(* CODESYS project PLC_CanIftHelper0.0.1.12.library
   Author: Cameron Johnson
   Placeholder: CanItfHelper
   Title: CanItfHelper
   Version: 0.0.1.12
   Description: This library has been supplied by Beckhoff Automation LLC As-Is and is intended only as an example implementation. Functionality is not guaranteed.
   Company: Beckhoff Automation LLC

Project tree, tasks and I/O mapping:
  libraries: Tc2_Standard, * (Beckhoff Automation GmbH); Tc2_System, * (Beckhoff Automation GmbH); Tc2_Utilities, * (Beckhoff Automation GmbH); Tc3_Module, * (Beckhoff Automation GmbH)
  11BitIdentifier/
    DUTs/
      data type ST_CanData_11bit
      data type ST_RxCanQueue_11bit
      data type ST_TxCanQueue_11bit
    POUs/
      function F_HwGetAddrInfo_11bit [ST]
      function F_HwSetAddrInfo_11bit [ST]
  29BitIdentifier/
    DUTs/
      data type ST_CanData_29bit
      data type ST_RxCanQueue_29bit
      data type ST_TxCanQueue_29bit
    POUs/
      function F_HwGetAddrInfo_29bit [ST]
      function F_HwSetAddrInfo_29bit [ST]
  29BitIdentifier_nTranscation/
    DUTs/
      data type ST_CanData_29bit_nTrans
      data type ST_RxCanQueue_29bit_nTrans
      data type ST_TxCanQueue_29bit_nTrans
    POUs/
      function F_HwGetAddrInfo_29bit_nTrans [ST]
      function F_HwSetAddrInfo_29bit_nTrans [ST]
  CanIftHelper/
    DUTs/
      data type E_CanItfHelperHResult
      data type ST_CanHeader
      data type ST_CanMsg
      data type U_RxQueue
      data type U_TxQueue
    POUs/
      function block FB_CanItfHelper [ST]: mCheckSetup, mRxMessageGet, mRxMessagesAck, mTxMessageAdd, mTxMessgesSend, mTxQueueReset
  DUTs/
    data type ST_CanMasterCycleInfo
    data type ST_CanMasterGlobalState
  GVLs/
    global variables GVL_CanItfHelper
    global variables Param_CanItfHelper
  Utilities/
    DUTs/
      data type E_CanRxMapperHResult
      data type ST_RxMapping
    POUs/
      function F_CanMessage_TO_CSV [ST]
      function F_CSV_TO_CanMessage [ST]
      function block FB_RxMapper [ST]: mAddMapping, mCheckSetup, mClearMappings, mCreateMsgMapping, mCreateNewMapping, mSetMappingCnt
  Version/
    global variables Global_Version
*)

// 11BitIdentifier/DUTs/ST_CanData_11bit
{attribute 'pack_mode' := '1'}
TYPE ST_CanData_11bit :
STRUCT
	nCobid: WORD; //bits 0-3 is CAN data length, bit 4 is CAN RTR flag, bit 5-15 is CAN Cobid.
	aData: ARRAY[0..7] OF BYTE;
END_STRUCT
END_TYPE

// 11BitIdentifier/DUTs/ST_RxCanQueue_11bit
{attribute 'pack_mode' := '1'}
TYPE ST_RxCanQueue_11bit :
STRUCT
	nTxCounter: UINT; // Tx handshake
	nRxCounter: UINT; // Rx handshake
	nNoOfmessages: UINT; // Number of messages relevent in Queue, ignore the rest.
	aMessages: ARRAY[0..GVL_CanItfHelper.nRxQueueUpperIndex] OF ST_CanData_11bit;
END_STRUCT
END_TYPE

// 11BitIdentifier/DUTs/ST_TxCanQueue_11bit
{attribute 'pack_mode' := '1'}
TYPE ST_TxCanQueue_11bit :
STRUCT
	nTxCounter: UINT; // Tx handshake
	nRxCounter: UINT; // Rx handshake
	nNoOfmessages: UINT; // Number of messages relevent in Queue, ignore the rest.
	aMessages: ARRAY[0..GVL_CanItfHelper.nTxQueueUpperIndex] OF ST_CanData_11bit;
END_STRUCT
END_TYPE

// 29BitIdentifier/DUTs/ST_CanData_29bit
{attribute 'pack_mode' := '1'}
TYPE ST_CanData_29bit :
STRUCT
	nLength: UINT; //values 0-8
	nCobid: DWORD; // bits0-28 CAN Cobid; bit 30 CAN RTR flag; bit 31 clear -> 11bit CAN Indentifier, set -> 29bit CAN Indentifier.
	aData: ARRAY[0..7] OF BYTE;
END_STRUCT
END_TYPE

// 29BitIdentifier/DUTs/ST_RxCanQueue_29bit
{attribute 'pack_mode' := '1'}
TYPE ST_RxCanQueue_29bit :
STRUCT
	nTxCounter: UINT; // Tx Handshake
	nRxCounter: UINT; // Rx handshake
	nNoOfmessages: UINT; // Number of messages relevent in Queue, ignore the rest.
	aMessages: ARRAY[0..GVL_CanItfHelper.nRxQueueUpperIndex] OF ST_CanData_29bit;
END_STRUCT
END_TYPE

// 29BitIdentifier/DUTs/ST_TxCanQueue_29bit
{attribute 'pack_mode' := '1'}
TYPE ST_TxCanQueue_29bit :
STRUCT
	nTxCounter: UINT; // Tx Handshake
	nRxCounter: UINT; // Rx handshake
	nNoOfmessages: UINT; // Number of messages relevent in Queue, ignore the rest.
	aMessages: ARRAY[0..GVL_CanItfHelper.nTxQueueUpperIndex] OF ST_CanData_29bit;
END_STRUCT
END_TYPE

// 29BitIdentifier_nTranscation/DUTs/ST_CanData_29bit_nTrans
{attribute 'pack_mode' := '1'}
TYPE ST_CanData_29bit_nTrans : //used with CX2500_M510 hardware
STRUCT
	ntransactionNumber : UINT; //unique identifier for message. See TxRxCanQueue.nTranactionNumber to see last TxMsg sent. Not used by FB_CanItfHelper.
	nLength: UINT; //values 0-8
	nCobid: DWORD; // bits0-28 CAN Cobid; bit 30 CAN RTR flag; bit 31 clear -> 11bit CAN Indentifier, set -> 29bit CAN Indentifier.
	aData: ARRAY[0..7] OF BYTE;
END_STRUCT
END_TYPE

// 29BitIdentifier_nTranscation/DUTs/ST_RxCanQueue_29bit_nTrans
{attribute 'pack_mode' := '1'}
TYPE ST_RxCanQueue_29bit_nTrans :
STRUCT
	nTxCounter: UINT; // Tx Handshake
	nRxCounter: UINT; // Rx handshake
	nNoOfmessages: UINT; // Number of messages relevent in Queue, ignore the rest.
	nTranactionNumber : UINT; // nTrans number of last sent TxMsg. Not used by FB_CanItfHelper.
	aMessages: ARRAY[0..GVL_CanItfHelper.nRxQueueUpperIndex] OF ST_CanData_29bit_nTrans;
END_STRUCT
END_TYPE

// 29BitIdentifier_nTranscation/DUTs/ST_TxCanQueue_29bit_nTrans
{attribute 'pack_mode' := '1'}
TYPE ST_TxCanQueue_29bit_nTrans :
STRUCT
	nTxCounter: UINT; 		// Tx Handshake
	nRxCounter: UINT; 		// Rx handshake
	nNoOfmessages: UINT; 	// Number of messages relevent in Queue, ignore the rest.
	nDummy : UINT;			//Reserved
	aMessages: ARRAY[0..GVL_CanItfHelper.nTxQueueUpperIndex] OF ST_CanData_29bit_nTrans;
END_STRUCT
END_TYPE

// CanIftHelper/DUTs/E_CanItfHelperHResult
{attribute 'qualified_only'}
{attribute 'strict'}
TYPE E_CanItfHelperHResult :
(
	NoError 						:= 0,  // values >= 0 implies no error and/or informational. values < 0 implies error. 
	NoError_11Bit					:= 1,
	NoError_29Bit					:= 2,
	NoError_29Bit_nTrans			:= 3,
	
	Error							:= -1, //Error, generic
	InvalidSetup 					:= -2, //pointers to ST_CanQueue are zero or sizeof ST_CanQueue doesn't equal 11bit or 29bit version.
	InvalidPointer					:= -3, //pointer parameter is zero.
	
	RxQueueHasUnreadMessages 		:= -100, // Rx Queue 'NoOfRxMessages' not equal RxMessagesAckedCnt, call either mGetRxMessages or mAckRxMessages.
	RxQueueEmpty 					:= -101, // Rx queue is empty, wait for more data.
	NoNewRxMessages 				:= -102, // Rx queue has not received new data yet.
	RxMessageInvalid				:= -103, // Rx Message returned is invalid, ignore result. Re-read Rx Messages.

	TxQueueFull 					:= -200, //NumOfMessages variable in Tx Queue is at or is greater then the allowed amount. Call aResetTxQueue and refill queue.
	TxQueueEmpty 					:= -201, // Tx queue 'NoOfTxMessages' value is zero, use mAddTxMessage to add messages.
	TxQueueInvalid					:= -202, //Tx Queue
	TxQueueIsBusy					:= -203 // Tx queue 'TxCounter' and Rx queue 'TxCounter' are not equal, waiting for CanInterface to send previous messages.
	
)DINT;
END_TYPE

// CanIftHelper/DUTs/ST_CanHeader
TYPE ST_CanHeader :
STRUCT
	nCobid: DWORD; // User level Cobid, use functions to handle bit mapping to CAN interface process data.
	bExtendedAddress: BOOL;// does nothing with 11bit version. Incorrectly 'cleared' does not cause errors and is automatically fixed.
	bRTR: BOOL; // Remote transmission request
	nMsgLength: UINT; // number of bytes in CAN message, values 0-8
END_STRUCT
END_TYPE

// CanIftHelper/DUTs/ST_CanMsg
TYPE ST_CanMsg :
STRUCT
	CanHeader: ST_CanHeader; // User level CAN header information.
	CanData: ARRAY[0..7] OF BYTE;
END_STRUCT
END_TYPE

// CanIftHelper/DUTs/U_RxQueue
{attribute 'hide'} 
TYPE U_RxQueue :
UNION
	pRxQueue_11bit 						: POINTER TO ST_RxCanQueue_11bit;
	pRxQueue_29bit 						: POINTER TO ST_RxCanQueue_29bit;
	pRxQueue_29bit_nTrans 				: POINTER TO ST_RxCanQueue_29bit_nTrans;
END_UNION
END_TYPE

// CanIftHelper/DUTs/U_TxQueue
{attribute 'hide'} 
TYPE U_TxQueue :
UNION
	pTxQueue_11bit 						: POINTER TO ST_TxCanQueue_11bit;
	pTxQueue_29bit 						: POINTER TO ST_TxCanQueue_29bit;
	pTxQueue_29bit_nTrans 				: POINTER TO ST_TxCanQueue_29bit_nTrans;
END_UNION
END_TYPE

// DUTs/ST_CanMasterCycleInfo
{attribute 'pack_mode' := '1'}
TYPE ST_CanMasterCycleInfo :
STRUCT
	 	{attribute 'hide'}
		_reserved1 : USINT;
		 {attribute 'hide'}
		_reserved2 : BIT;
		 {attribute 'hide'}
		_reserved3 : BIT;
		 {attribute 'hide'}
		_reserved4 : BIT;
		 {attribute 'hide'}
		_reserved5 : BIT;
	deviceDiag : BIT; // 1 = Diagnosis Data changed, use ADS-Read (Port 200, Index-Group 0xF100) to get the data
	syncError : BIT;//  reserved for future use
	cycleToggle : BIT;// toggles with every cycle
	cycleError : BIT;//  1 = at least one CANopen Slave has a NodeState unequal zero
	cycleCounter : UINT;//  EL6751 increments this counter once when the cycle is finished and the the EtherCAT Input Data were updated
	error : USINT;// indicates the number of CANopen slaves with a NodeState unequal zero
		 {attribute 'hide'}
		_reserved6 : USINT;
	actualCycleTime : UINT;//  indicates the actual Cycle-Time
END_STRUCT
END_TYPE

// DUTs/ST_CanMasterGlobalState
{attribute 'pack_mode' := '1'}
TYPE ST_CanMasterGlobalState :
STRUCT
	DeviceState : UINT;(*  0: Device is in state RUN,  1: Device is in state RESET,  2: Device is in state OFFLINE,  3: Device is in state STOP*)
	RxErrorCounter	: USINT;(* RxError-Counter of the CAN-Controller*)
	TxErrorCounter : USINT; (*TxError-Counter of the CAN-Controller*)
	CanControllerBUSOFF : BIT;
	CanControllerWarningLimit : BIT;
	RxQueueOverrun : BIT;
	HiPrioTxQueueOverrun : BIT;
	LoPrioTxQueueOverrun : BIT;
	CanSendError : BIT;
		{attribute 'hide'}
		_reserved6 : BIT;
		{attribute 'hide'}
		_reserved7 : BIT;
		{attribute 'hide'}
		_reserved8 : BIT;
		{attribute 'hide'}
		_reserved9 : BIT;
		{attribute 'hide'}
		_reserved10 : BIT;
		{attribute 'hide'}
		_reserved11 : BIT;
		{attribute 'hide'}
		_reserved12 : BIT;
		{attribute 'hide'}
		_reserved13 : BIT;
		{attribute 'hide'}
		_reserved14 : BIT;
	SyncMsgToggle : BIT; // toggles with every SYNC message sent
	BusLoad : UINT; // value in perecent [%]
END_STRUCT
END_TYPE

// Utilities/DUTs/E_CanRxMapperHResult
{attribute 'qualified_only'}
{attribute 'strict'}
TYPE E_CanRxMapperHResult :
(
	NoError := 0,
	
	RxMapperHasInvalidSetup			:= -1, // pCanItfHelper or nCanItfHelperSize parameters are invalid. 
	CanHelperSetupIsInvalid			:= -2, // FB_CanItfHelper.bValidSetup = false
	MappingSetupIsInvalid			:= -3, // paMappingData or nMappingDataSize parameters are invalid.
	
	InvalidParameter				:= -10, //generic error call parameters.
	
	RxMappingsListFull				:= -100, // nAddMappingIndex > GVL_CanItfHelper.nRxMapperUpperIndex, increase mapping list size, clear list and re-add and/or use another instance.
	
	
	RxMappingDestSizeError			:= -200, // destination size is either size or is error causing size.
	RxMappingDestPointerError		:= -201, // destination pointer is zero.
	
	//info / warnings
	RxMappingNotRunning				:= 1, // Rx mapping bRun is false.
	RxMappingHasError				:= 2 // FB_RxPdoMapper has a ST_RxPdoMapping in array aMappingData with an error. Fix issue and toggle bRun bit in ST_RxPdoMapping to clear error.			


)DINT;
END_TYPE

// Utilities/DUTs/ST_RxMapping
TYPE ST_RxMapping :
STRUCT
	i_bRun				: BOOL; // Mapping is ignored if set false.
	i_stCanMsg			: ST_CanMsg; // See CAN header informaiton for information rx mapper checks against. If MsgLength is less then i_cbDestSize return data is allow.
	i_pDestAddr			: POINTER TO BYTE; // Make sure pointers are valid before calling mapper! You may have to detect online changes and re-initalize mapping info.
	i_cbDestSize		: UDINT;// byte size of destination variable.
	o_nUpdateCount		: UINT; // If pointer and/or destsize parameters are incorrect, this value will still update. Increments if Cobid, flags ExtenedAddress and RTR is valid.	
	o_bBusy				: BOOL; // is true is data from recieved message is copied. 
	o_bError			: BOOL; // true is an input parameter would prevent data from recieved message to be copied. 
END_STRUCT
END_TYPE

// GVLs/GVL_CanItfHelper
{attribute 'qualified_only' := ''}
{attribute 'global_init_slot' := '110'}
VAR_GLOBAL CONSTANT
	nTxQueueUpperIndex		: UINT := (Param_CanItfHelper.nTxQueueSize - 1);// size of send queue minus 1, upper array index
	nRxQueueUpperIndex		: UINT := (Param_CanItfHelper.nRxQueueSize - 1);// size of receive queue minus 1, upper array index
END_VAR

// GVLs/Param_CanItfHelper
{attribute 'global_init_slot' := '100'}
{attribute 'qualified_only' := ''}
{attribute 'parameterlist' := ''}
VAR_GLOBAL CONSTANT
	nTxQueueSize			: UINT := 10; // number of messages in Tx queue.
	nRxQueueSize			: UINT := 10;// number of messages in Rx queue.
	sCSV_deliminator		: STRING(2) := ','; // deliminator used in CSV functions.
END_VAR

// Version/Global_Version
{attribute 'TcGenerated'}
{attribute 'no-analysis'}
{attribute 'linkalways'}
// This function has been automatically generated from the project information.
VAR_GLOBAL CONSTANT
	{attribute 'const_non_replaced'}
	stLibVersion_CanItfHelper : ST_LibVersion := (iMajor := 0, iMinor := 0, iBuild := 1, iRevision := 12, nFlags := 0, sVersion := '0.0.1.12');
END_VAR

// 11BitIdentifier/POUs/F_HwGetAddrInfo_11bit
{attribute 'hide'}
FUNCTION F_HwGetAddrInfo_11bit : ST_CanHeader//function to map cobid, RTR and datalength to ST_CanHeader.
VAR_INPUT
	nInput: WORD;// bit 0-3 datalength, bit4 RTR, bit 5-16 Cobid
END_VAR

F_HwGetAddrInfo_11bit.nCobid := WORD_TO_DWORD( 16#7FF AND SHR(nInput,5)); //shift cobid from 5-16 to bits 0-10, limits cobid to max value

F_HwGetAddrInfo_11bit.bRTR := nInput.4; // gets RTR bit

F_HwGetAddrInfo_11bit.bExtendedAddress := FALSE; // 29bit is not used, set false;

IF ((nInput AND 16#F) > 8) THEN // returns the first bits 0-3 which is data length value, checks to make sure length is not greater than max data length (8);
	F_HwGetAddrInfo_11bit.nMsgLength := 8;//issue getting data length, set to max.
ELSE
	F_HwGetAddrInfo_11bit.nMsgLength := (nInput AND 16#F);// returns the first bits 0-3 which is data length value
END_IF

END_FUNCTION

// 11BitIdentifier/POUs/F_HwSetAddrInfo_11bit
{attribute 'hide'}
FUNCTION F_HwSetAddrInfo_11bit : WORD
VAR_INPUT
	stInput: ST_CanHeader;
END_VAR

F_HwSetAddrInfo_11bit := SHL((16#7FF AND DWORD_TO_WORD(stInput.nCobid)),5); //shift cobid from 0-10 to bits 5-16, limits cobid to max value

F_HwSetAddrInfo_11bit.4 := stInput.bRTR;// gets RTR bit

IF (stInput.nMsgLength > 8) THEN// returns the first bits 0-3 which is data length value, checks to make sure length is not greater than max data length (8);
	F_HwSetAddrInfo_11bit := 8;//issue getting data length, set to max.
ELSE
	F_HwSetAddrInfo_11bit :=  F_HwSetAddrInfo_11bit OR UINT_TO_WORD(stInput.nMsgLength);// sets bits 0-3 which is can data length. 
END_IF

//Extended Indentifier isn't used.

END_FUNCTION

// 29BitIdentifier/POUs/F_HwGetAddrInfo_29bit
{attribute 'hide'}
FUNCTION F_HwGetAddrInfo_29bit : ST_CanHeader
VAR_INPUT
	stInput: ST_CanData_29bit;
END_VAR

F_HwGetAddrInfo_29bit.nCobid := 16#3FFFFFFF AND UDINT_TO_DWORD(stInput.nCobid);// limits cobid to max value

F_HwGetAddrInfo_29bit.bRTR := stInput.nCobid.30;// gets RTR bit

F_HwGetAddrInfo_29bit.bExtendedAddress := stInput.nCobid.31;//gets extended address flag, if set raw can message had 29bit for identification on the wire.

IF (stInput.nLength > 8) THEN
	F_HwGetAddrInfo_29bit.nMsgLength := 8;
ELSE
	F_HwGetAddrInfo_29bit.nMsgLength := stInput.nLength;
END_IF

END_FUNCTION

// 29BitIdentifier/POUs/F_HwSetAddrInfo_29bit
{attribute 'hide'}
FUNCTION F_HwSetAddrInfo_29bit : ST_CanData_29bit
VAR_INPUT
	stInput: ST_CanHeader;
END_VAR

F_HwSetAddrInfo_29bit.nCobid := 16#3FFFFFFF AND stInput.nCobid;

IF (stInput.nCobid > 16#7FF AND NOT stInput.bExtendedAddress) THEN // check cobid and extended address flags is set correctly
	stInput.bExtendedAddress := TRUE;//fix issue
END_IF

F_HwSetAddrInfo_29bit.nCobid.31 := stInput.bExtendedAddress;//sets extended address flag, if set raw can message will have 29bit for identification on the wire.

F_HwSetAddrInfo_29bit.nCobid.30 := stInput.bRTR;// sets RTR bit

IF (stInput.nMsgLength > 8) THEN
	F_HwSetAddrInfo_29bit.nLength := 8;
ELSE
	F_HwSetAddrInfo_29bit.nLength := stInput.nMsgLength;
END_IF

END_FUNCTION

// 29BitIdentifier_nTranscation/POUs/F_HwGetAddrInfo_29bit_nTrans
{attribute 'hide'}
FUNCTION F_HwGetAddrInfo_29bit_nTrans : ST_CanHeader
VAR_INPUT
	stInput: ST_CanData_29bit_nTrans;
END_VAR

F_HwGetAddrInfo_29bit_nTrans.nCobid := 16#3FFFFFFF AND UDINT_TO_DWORD(stInput.nCobid);// limits cobid to max value

F_HwGetAddrInfo_29bit_nTrans.bRTR := stInput.nCobid.30;// gets RTR bit

F_HwGetAddrInfo_29bit_nTrans.bExtendedAddress := stInput.nCobid.31;//gets extended address flag, if set raw can message had 29bit for identification on the wire.

IF (stInput.nLength > 8) THEN
	F_HwGetAddrInfo_29bit_nTrans.nMsgLength := 8;
ELSE
	F_HwGetAddrInfo_29bit_nTrans.nMsgLength := stInput.nLength;
END_IF

END_FUNCTION

// 29BitIdentifier_nTranscation/POUs/F_HwSetAddrInfo_29bit_nTrans
{attribute 'hide'}
FUNCTION F_HwSetAddrInfo_29bit_nTrans : ST_CanData_29bit_nTrans
VAR_INPUT
	stInput: ST_CanHeader;
END_VAR

F_HwSetAddrInfo_29bit_nTrans.nCobid := 16#3FFFFFFF AND stInput.nCobid;

IF (stInput.nCobid > 16#7FF AND NOT stInput.bExtendedAddress) THEN // check cobid and extended address flags is set correctly
	stInput.bExtendedAddress := TRUE;//fix issue
END_IF

F_HwSetAddrInfo_29bit_nTrans.nCobid.31 := stInput.bExtendedAddress;//sets extended address flag, if set raw can message will have 29bit for identification on the wire.

F_HwSetAddrInfo_29bit_nTrans.nCobid.30 := stInput.bRTR;// sets RTR bit

IF (stInput.nMsgLength > 8) THEN
	F_HwSetAddrInfo_29bit_nTrans.nLength := 8;
ELSE
	F_HwSetAddrInfo_29bit_nTrans.nLength := stInput.nMsgLength;
END_IF

END_FUNCTION

// CanIftHelper/POUs/FB_CanItfHelper
{attribute 'hide_all_locals'}
FUNCTION_BLOCK FB_CanItfHelper //Call FB once per task tick before calling methods.
VAR_INPUT
	pRxQueue 				: POINTER TO BYTE; //must pass either ST_RxCanQueue_11bit or ST_RxCanQueue_29bit or ST_RxCanQueue_29bit_CX2500_M510
	cbRxQueueSize 			: UDINT;
	pTxQueue 				: POINTER TO BYTE; //must pass either ST_TxCanQueue_11bit or ST_TxCanQueue_29bit or ST_TxCanQueue_29bit_CX2500_M510
	cbTxQueueSize 			: UDINT;	
END_VAR
VAR_OUTPUT
	bValidSetup				: BOOL := FALSE;// indictor that input pointers are non zero and sizes are correct.
	bRxMsgsAcked			: BOOL;// RxMessages have been acknowledge, RxQueue will update automatically when next RxMessage/s is received.
	bTxMsgsSending			: BOOL;// TxMessages have been flagged to be sent the next time an IO update occurs.
END_VAR

VAR
	_uRxQueue				: U_RxQueue;
	_uTxQueue				: U_TxQueue;
	
	_nTxSendTaskCnt			: UDINT; //Internal counter helps determine if mAddTxMessage is allowed to add more messages even though TxQueue. TxCounter is flagged to send new data. Intended to optimism Queue by enlimiting a race condition. 
	_nRxMsgReadedIndex 		: UINT; 
	_nTxMsgSendCnt 			: UINT;
	_bTxMsgSent				: BOOL;
END_VAR

THIS^.mCheckSetup();

METHOD PRIVATE mCheckSetup : E_CanItfHelperHResult
VAR

END_VAR
mCheckSetup := E_CanItfHelperHResult.NoError;
	
IF (pRxQueue = NULL) AND (pTxQueue = NULL) THEN
	bValidSetup := FALSE;
	mCheckSetup := E_CanItfHelperHResult.InvalidSetup;
	RETURN;
END_IF	

IF cbRxQueueSize =  SIZEOF(ST_RxCanQueue_11bit) AND cbTxQueueSize = SIZEOF(ST_TxCanQueue_11bit) THEN
	mCheckSetup := E_CanItfHelperHResult.NoError_11Bit;
ELSIF cbRxQueueSize =  SIZEOF(ST_RxCanQueue_29bit) AND cbTxQueueSize = SIZEOF(ST_TxCanQueue_29bit) THEN
	mCheckSetup := E_CanItfHelperHResult.NoError_29Bit;
ELSIF cbRxQueueSize =  SIZEOF(ST_RxCanQueue_29bit_nTrans) AND cbTxQueueSize = SIZEOF(ST_TxCanQueue_29bit_nTrans) THEN
	mCheckSetup := E_CanItfHelperHResult.NoError_29Bit_nTrans;
ELSE 
	mCheckSetup := E_CanItfHelperHResult.Error;
END_IF

IF mCheckSetup <> E_CanItfHelperHResult.Error THEN
	bValidSetup := TRUE;
	_uRxQueue.pRxQueue_11bit := pRxQueue;
	_uTxQueue.pTxQueue_11bit := pTxQueue;
ELSE
	bValidSetup := FALSE;
	mCheckSetup := E_CanItfHelperHResult.InvalidSetup;
	RETURN;
END_IF
END_METHOD

METHOD mRxMessageGet : E_CanItfHelperHResult //Copies the top in the RxQueue to a ST_CanMessage.
VAR_INPUT
	pRxCanMessage : POINTER TO ST_CanMsg := NULL; //Gets current CAN message on the next message in queue and overwrites value passed by reference stCanMsg, must pass type ST_CanMessage
	bPeakOnly : BOOL := FALSE; // if true and method completes successfully -> message is not from RxQueue. 	 
END_VAR
mRxMessageGet := THIS^.mCheckSetup();
IF (mRxMessageGet <= E_CanItfHelperHResult.Error) THEN
	RETURN;
END_IF

IF (pRxCanMessage = NULL) THEN
	mRxMessageGet := E_CanItfHelperHResult.InvalidPointer;
	RETURN;
END_IF


CASE mRxMessageGet OF
	E_CanItfHelperHResult.NoError_11Bit:	//Checks fors 11bit items
		IF (_uRxQueue.pRxQueue_11bit^.nNoOfmessages > GVL_CanItfHelper.nRxQueueUpperIndex) THEN
			mRxMessageGet := E_CanItfHelperHResult.RxMessageInvalid;
			RETURN;
		END_IF
		
		IF (_uRxQueue.pRxQueue_11bit^.nNoOfmessages = _nRxMsgReadedIndex) OR bRxMsgsAcked THEN
			mRxMessageGet := E_CanItfHelperHResult.RxQueueEmpty;
			RETURN;
		END_IF
		
		IF (_uRxQueue.pRxQueue_11bit^.nRxCounter <> _uTxQueue.pTxQueue_11bit^.nRxCounter) THEN
			IF bRxMsgsAcked THEN
				_nRxMsgReadedIndex := 0;
			END_IF
			bRxMsgsAcked := FALSE;
		END_IF
		
		pRxCanMessage^.CanData := _uRxQueue.pRxQueue_11bit^.aMessages[_nRxMsgReadedIndex MOD Param_CanItfHelper.nRxQueueSize].aData;
		pRxCanMessage^.CanHeader := F_HwGetAddrInfo_11bit(nInput := _uRxQueue.pRxQueue_11bit^.aMessages[_nRxMsgReadedIndex MOD Param_CanItfHelper.nRxQueueSize].nCobid);
		mRxMessageGet := E_CanItfHelperHResult.NoError;
		
		IF NOT bPeakOnly THEN
			_nRxMsgReadedIndex := _nRxMsgReadedIndex + 1;
		END_IF
		
	E_CanItfHelperHResult.NoError_29Bit:	//Checks for 29 bit items
	
		IF (_uRxQueue.pRxQueue_29bit^.nNoOfmessages > GVL_CanItfHelper.nRxQueueUpperIndex) THEN
			mRxMessageGet := E_CanItfHelperHResult.RxMessageInvalid;
			RETURN;
		END_IF
		
		IF (_uRxQueue.pRxQueue_29bit^.nNoOfmessages = _nRxMsgReadedIndex) OR bRxMsgsAcked THEN
			mRxMessageGet := E_CanItfHelperHResult.RxQueueEmpty;
			RETURN;
		END_IF
		
		IF (_uRxQueue.pRxQueue_29bit^.nRxCounter <> _uTxQueue.pTxQueue_29bit^.nRxCounter) THEN
			IF bRxMsgsAcked THEN
				_nRxMsgReadedIndex := 0;
			END_IF
			bRxMsgsAcked := FALSE;
		END_IF
		
		pRxCanMessage^.CanData := _uRxQueue.pRxQueue_29bit^.aMessages[_nRxMsgReadedIndex MOD Param_CanItfHelper.nRxQueueSize].aData;
		pRxCanMessage^.CanHeader := F_HwGetAddrInfo_29bit(stInput := _uRxQueue.pRxQueue_29bit^.aMessages[_nRxMsgReadedIndex MOD Param_CanItfHelper.nRxQueueSize]);
		mRxMessageGet := E_CanItfHelperHResult.NoError;
		
		IF NOT bPeakOnly THEN
			_nRxMsgReadedIndex := _nRxMsgReadedIndex + 1;
		END_IF
		
	E_CanItfHelperHResult.NoError_29Bit_nTrans: 	//Checks for 29 bit items
		
		IF (_uRxQueue.pRxQueue_29bit_nTrans^.nNoOfmessages > GVL_CanItfHelper.nRxQueueUpperIndex) THEN
			mRxMessageGet := E_CanItfHelperHResult.RxMessageInvalid;
			RETURN;
		END_IF
		
		IF (_uRxQueue.pRxQueue_29bit_nTrans^.nNoOfmessages = _nRxMsgReadedIndex) OR bRxMsgsAcked THEN
			mRxMessageGet := E_CanItfHelperHResult.RxQueueEmpty;
			RETURN;
		END_IF
		
		IF (_uRxQueue.pRxQueue_29bit_nTrans^.nRxCounter <> _uTxQueue.pTxQueue_29bit_nTrans^.nRxCounter) THEN
			IF bRxMsgsAcked THEN
				_nRxMsgReadedIndex := 0;
			END_IF
			bRxMsgsAcked := FALSE;
		END_IF
		
		pRxCanMessage^.CanData := _uRxQueue.pRxQueue_29bit_nTrans^.aMessages[_nRxMsgReadedIndex MOD Param_CanItfHelper.nRxQueueSize].aData;
		pRxCanMessage^.CanHeader := F_HwGetAddrInfo_29bit_nTrans(stInput := _uRxQueue.pRxQueue_29bit_nTrans^.aMessages[_nRxMsgReadedIndex MOD Param_CanItfHelper.nRxQueueSize]);
		mRxMessageGet := E_CanItfHelperHResult.NoError;
		
		IF NOT bPeakOnly THEN
			_nRxMsgReadedIndex := _nRxMsgReadedIndex + 1;
		END_IF
	
END_CASE
END_METHOD

METHOD mRxMessagesAck : E_CanItfHelperHResult //ackownledge current RxMessages to new RxMessages to be recieved. NOTE: Call this at the end of the PLC task cycle.
VAR_INPUT
	bForceAck : BOOL;	//If true, RxQueue is ackownledged even if there are un read messages.
END_VAR
mRxMessagesAck := THIS^.mCheckSetup();
IF (mRxMessagesAck <= E_CanItfHelperHResult.Error) THEN
	RETURN;
END_IF

CASE mRxMessagesAck OF 
	E_CanItfHelperHResult.NoError_11Bit:
		IF (_uRxQueue.pRxQueue_11bit^.nRxCounter <> _uTxQueue.pTxQueue_11bit^.nRxCounter) THEN
	
			IF ((_uRxQueue.pRxQueue_11bit^.nNoOfmessages = _nRxMsgReadedIndex) OR (bForceAck = TRUE)) THEN
				_uTxQueue.pTxQueue_11bit^.nRxCounter := _uRxQueue.pRxQueue_11bit^.nRxCounter;
				_nRxMsgReadedIndex := 0;
				bRxMsgsAcked := TRUE;
				mRxMessagesAck := E_CanItfHelperHResult.NoError;
			ELSE
				bRxMsgsAcked := FALSE;
				mRxMessagesAck := E_CanItfHelperHResult.RxQueueHasUnreadMessages;
			END_IF
			
		ELSE	
			_nRxMsgReadedIndex := 0;
			bRxMsgsAcked := TRUE;
			mRxMessagesAck :=	E_CanItfHelperHResult.NoNewRxMessages;
		END_IF
	
	E_CanItfHelperHResult.NoError_29Bit:	//29bit handling
		IF (_uRxQueue.pRxQueue_29bit^.nRxCounter <> _uTxQueue.pTxQueue_29bit^.nRxCounter) THEN
	
			IF ((_uRxQueue.pRxQueue_29bit^.nNoOfmessages = _nRxMsgReadedIndex) OR (bForceAck = TRUE)) THEN
				_uTxQueue.pTxQueue_29bit^.nRxCounter := _uRxQueue.pRxQueue_29bit^.nRxCounter;
				_nRxMsgReadedIndex := 0;
				bRxMsgsAcked := TRUE;
				mRxMessagesAck := E_CanItfHelperHResult.NoError;
			ELSE
				bRxMsgsAcked := FALSE;
				mRxMessagesAck := E_CanItfHelperHResult.RxQueueHasUnreadMessages;
			END_IF
			
		ELSE	
			_nRxMsgReadedIndex := 0;
			bRxMsgsAcked := TRUE;
			mRxMessagesAck :=	E_CanItfHelperHResult.NoNewRxMessages;
		END_IF
	
	E_CanItfHelperHResult.NoError_29Bit_nTrans:	//29bit handling
		IF (_uRxQueue.pRxQueue_29bit_nTrans^.nRxCounter <> _uTxQueue.pTxQueue_29bit_nTrans^.nRxCounter) THEN
	
			IF ((_uRxQueue.pRxQueue_29bit_nTrans^.nNoOfmessages = _nRxMsgReadedIndex) OR (bForceAck = TRUE)) THEN
				_uTxQueue.pTxQueue_29bit_nTrans^.nRxCounter := _uRxQueue.pRxQueue_29bit_nTrans^.nRxCounter;
				_nRxMsgReadedIndex := 0;
				bRxMsgsAcked := TRUE;
				mRxMessagesAck := E_CanItfHelperHResult.NoError;
			ELSE
				bRxMsgsAcked := FALSE;
				mRxMessagesAck := E_CanItfHelperHResult.RxQueueHasUnreadMessages;
			END_IF
			
		ELSE	
			_nRxMsgReadedIndex := 0;
			bRxMsgsAcked := TRUE;
			mRxMessagesAck :=	E_CanItfHelperHResult.NoNewRxMessages;
			_nRxMsgReadedIndex := 0;
		END_IF
	ELSE
		mRxMessagesAck := E_CanItfHelperHResult.InvalidSetup;
END_CASE
END_METHOD

METHOD mTxMessageAdd : E_CanItfHelperHResult
VAR_INPUT
	pTxCanMessage : POINTER TO ST_CanMsg := NULL; //Writes stCanQueue to queue, value passed by reference, must pass type ST_CanMessage
END_VAR
mTxMessageAdd := THIS^.mCheckSetup();
IF (mTxMessageAdd < E_CanItfHelperHResult.NoError) THEN
	RETURN;
END_IF

IF (pTxCanMessage = NULL) THEN
	mTxMessageAdd := E_CanItfHelperHResult.InvalidPointer;
	RETURN;
END_IF


//Add Case here
CASE mTxMessageAdd OF
	E_CanItfHelperHResult.NoError_11Bit:

		IF (_uTxQueue.pTxQueue_11bit^.nTxCounter <> _uRxQueue.pRxQueue_11bit^.nTxCounter) THEN
			IF (_nTxSendTaskCnt <> TwinCAT_SystemInfoVarList._TaskInfo[GETCURTASKINDEXEX()].CycleCount) THEN
				mTxMessageAdd := E_CanItfHelperHResult.TxQueueIsBusy;
				RETURN;
			END_IF
		END_IF
	
		IF _bTxMsgSent AND (_nTxSendTaskCnt <> TwinCAT_SystemInfoVarList._TaskInfo[GETCURTASKINDEXEX()].CycleCount) THEN
			_nTxMsgSendCnt := 0;
			_bTxMsgSent := FALSE;
		END_IF
		
		IF (_nTxMsgSendCnt > GVL_CanItfHelper.nTxQueueUpperIndex) THEN
			mTxMessageAdd := E_CanItfHelperHResult.TxQueueFull;
			RETURN;
		END_IF	
	

		_uTxQueue.pTxQueue_11bit^.aMessages[_nTxMsgSendCnt].nCobid := F_HwSetAddrInfo_11bit(pTxCanMessage^.CanHeader);
		_uTxQueue.pTxQueue_11bit^.aMessages[_nTxMsgSendCnt].aData := pTxCanMessage^.CanData;
		_nTxMsgSendCnt := _nTxMsgSendCnt + 1;
		mTxMessageAdd := E_CanItfHelperHResult.NoError;
		
	E_CanItfHelperHResult.NoError_29Bit:
		
		IF (_uTxQueue.pTxQueue_29bit^.nTxCounter <> _uRxQueue.pRxQueue_29bit^.nTxCounter) THEN
			IF (_nTxSendTaskCnt <> TwinCAT_SystemInfoVarList._TaskInfo[GETCURTASKINDEXEX()].CycleCount) THEN
				mTxMessageAdd := E_CanItfHelperHResult.TxQueueIsBusy;
				RETURN;
			END_IF
		END_IF
	
		IF _bTxMsgSent AND (_nTxSendTaskCnt <> TwinCAT_SystemInfoVarList._TaskInfo[GETCURTASKINDEXEX()].CycleCount) THEN
			_nTxMsgSendCnt := 0;
			_bTxMsgSent := FALSE;
		END_IF
		
		IF (_nTxMsgSendCnt > GVL_CanItfHelper.nTxQueueUpperIndex) THEN
			mTxMessageAdd := E_CanItfHelperHResult.TxQueueFull;
			RETURN;
		END_IF
		
	
		_uTxQueue.pTxQueue_29bit^.aMessages[_nTxMsgSendCnt] := F_HwSetAddrInfo_29bit(pTxCanMessage^.CanHeader);
		_uTxQueue.pTxQueue_29bit^.aMessages[_nTxMsgSendCnt].aData := pTxCanMessage^.CanData;
		_nTxMsgSendCnt := _nTxMsgSendCnt + 1;
		mTxMessageAdd := E_CanItfHelperHResult.NoError;
	
	
	E_CanItfHelperHResult.NoError_29Bit_nTrans:
	
		IF (_uTxQueue.pTxQueue_29bit_nTrans^.nTxCounter <> _uRxQueue.pRxQueue_29bit_nTrans^.nTxCounter) THEN
			IF (_nTxSendTaskCnt <> TwinCAT_SystemInfoVarList._TaskInfo[GETCURTASKINDEXEX()].CycleCount) THEN
				mTxMessageAdd := E_CanItfHelperHResult.TxQueueIsBusy;
				RETURN;
			END_IF
		END_IF
	
		IF _bTxMsgSent AND (_nTxSendTaskCnt <> TwinCAT_SystemInfoVarList._TaskInfo[GETCURTASKINDEXEX()].CycleCount) THEN
			_nTxMsgSendCnt := 0;
			_bTxMsgSent := FALSE;
		END_IF
		
		IF (_nTxMsgSendCnt > GVL_CanItfHelper.nTxQueueUpperIndex) THEN
			mTxMessageAdd := E_CanItfHelperHResult.TxQueueFull;
			RETURN;
		END_IF
		
		_uTxQueue.pTxQueue_29bit_nTrans^.aMessages[_nTxMsgSendCnt] := F_HwSetAddrInfo_29bit_nTrans(pTxCanMessage^.CanHeader);
		_uTxQueue.pTxQueue_29bit_nTrans^.aMessages[_nTxMsgSendCnt].aData := pTxCanMessage^.CanData;
		_nTxMsgSendCnt := _nTxMsgSendCnt + 1;
		mTxMessageAdd := E_CanItfHelperHResult.NoError;
END_CASE
END_METHOD

METHOD mTxMessgesSend : E_CanItfHelperHResult
mTxMessgesSend := THIS^.mCheckSetup();
IF (mTxMessgesSend < E_CanItfHelperHResult.NoError) THEN
	RETURN;
END_IF

CASE mTxMessgesSend OF
	E_CanItfHelperHResult.NoError_11Bit:

		IF (_uTxQueue.pTxQueue_11bit^.nNoOfmessages > Param_CanItfHelper.nTxQueueSize) THEN
			_nTxMsgSendCnt := GVL_CanItfHelper.nTxQueueUpperIndex;
			mTxMessgesSend := E_CanItfHelperHResult.TxQueueInvalid;
			RETURN;
		END_IF	
		
		IF (_uTxQueue.pTxQueue_11bit^.nTxCounter <> _uRxQueue.pRxQueue_11bit^.nTxCounter)THEN
			IF (_nTxSendTaskCnt <> TwinCAT_SystemInfoVarList._TaskInfo[GETCURTASKINDEXEX()].CycleCount) THEN
				mTxMessgesSend := E_CanItfHelperHResult.TxQueueIsBusy;
				RETURN;
			END_IF
		END_IF	
		
		(*(pTxQueue_11bit^.nTxCounter = pRxQueue_11bit^.nTxCounter)*)
		IF _bTxMsgSent AND (_nTxSendTaskCnt <> TwinCAT_SystemInfoVarList._TaskInfo[GETCURTASKINDEXEX()].CycleCount) THEN
			mTxMessgesSend := E_CanItfHelperHResult.TxQueueEmpty;
			_nTxMsgSendCnt := 0;
			_bTxMsgSent := FALSE;
			RETURN;
		END_IF
		
		
		(*(pTxQueue_11bit^.nTxCounter = pRxQueue_11bit^.nTxCounter)*)
		_uTxQueue.pTxQueue_11bit^.nTxCounter := _uRxQueue.pRxQueue_11bit^.nTxCounter + 1;
		_uTxQueue.pTxQueue_11bit^.nNoOfmessages := _nTxMsgSendCnt;
		_bTxMsgSent := TRUE;
		_nTxSendTaskCnt := TwinCAT_SystemInfoVarList._TaskInfo[GETCURTASKINDEXEX()].CycleCount;
		mTxMessgesSend := E_CanItfHelperHResult.NoError;
		
	E_CanItfHelperHResult.NoError_29Bit:
		IF (_uTxQueue.pTxQueue_29bit^.nNoOfmessages > Param_CanItfHelper.nTxQueueSize) THEN
			_nTxMsgSendCnt := GVL_CanItfHelper.nTxQueueUpperIndex;
			mTxMessgesSend := E_CanItfHelperHResult.TxQueueInvalid;
			RETURN;
		END_IF	
		
		IF (_uTxQueue.pTxQueue_29bit^.nTxCounter <> _uRxQueue.pRxQueue_29bit^.nTxCounter)THEN
			IF (_nTxSendTaskCnt <> TwinCAT_SystemInfoVarList._TaskInfo[GETCURTASKINDEXEX()].CycleCount) THEN
				mTxMessgesSend := E_CanItfHelperHResult.TxQueueIsBusy;
				RETURN;
			END_IF
		END_IF	
		
		IF _bTxMsgSent AND (_nTxSendTaskCnt <> TwinCAT_SystemInfoVarList._TaskInfo[GETCURTASKINDEXEX()].CycleCount) THEN
			mTxMessgesSend := E_CanItfHelperHResult.TxQueueEmpty;
			_nTxMsgSendCnt := 0;
			_bTxMsgSent := FALSE;
			RETURN;
		END_IF
		
		_uTxQueue.pTxQueue_29bit^.nTxCounter := _uRxQueue.pRxQueue_29bit^.nTxCounter + 1;
		_uTxQueue.pTxQueue_29bit^.nNoOfmessages := _nTxMsgSendCnt;
		_bTxMsgSent := TRUE;
		_nTxSendTaskCnt := TwinCAT_SystemInfoVarList._TaskInfo[GETCURTASKINDEXEX()].CycleCount;
		mTxMessgesSend := E_CanItfHelperHResult.NoError;
		
	E_CanItfHelperHResult.NoError_29Bit_nTrans:
		IF (_uTxQueue.pTxQueue_29bit_nTrans^.nNoOfmessages > Param_CanItfHelper.nTxQueueSize) THEN
			_nTxMsgSendCnt := GVL_CanItfHelper.nTxQueueUpperIndex;
			mTxMessgesSend := E_CanItfHelperHResult.TxQueueInvalid;
			RETURN;
		END_IF	
		
		IF (_uTxQueue.pTxQueue_29bit_nTrans^.nTxCounter <> _uRxQueue.pRxQueue_29bit_nTrans^.nTxCounter)THEN
			IF (_nTxSendTaskCnt <> TwinCAT_SystemInfoVarList._TaskInfo[GETCURTASKINDEXEX()].CycleCount) THEN
				mTxMessgesSend := E_CanItfHelperHResult.TxQueueIsBusy;
				RETURN;
			END_IF
		END_IF	
		
		IF _bTxMsgSent AND (_nTxSendTaskCnt <> TwinCAT_SystemInfoVarList._TaskInfo[GETCURTASKINDEXEX()].CycleCount) THEN
			mTxMessgesSend := E_CanItfHelperHResult.TxQueueEmpty;
			_nTxMsgSendCnt := 0;
			_bTxMsgSent := FALSE;
			RETURN;
		END_IF
		
		_uTxQueue.pTxQueue_29bit_nTrans^.nTxCounter := _uRxQueue.pRxQueue_29bit_nTrans^.nTxCounter + 1;
		_uTxQueue.pTxQueue_29bit_nTrans^.nNoOfmessages := _nTxMsgSendCnt;
		_bTxMsgSent := TRUE;
		_nTxSendTaskCnt := TwinCAT_SystemInfoVarList._TaskInfo[GETCURTASKINDEXEX()].CycleCount;
		mTxMessgesSend := E_CanItfHelperHResult.NoError;
END_CASE

bTxMsgsSending := _bTxMsgSent;
END_METHOD

METHOD mTxQueueReset : E_CanItfHelperHResult
mTxQueueReset := THIS^.mCheckSetup();
IF (mTxQueueReset < E_CanItfHelperHResult.NoError) THEN
	RETURN;
END_IF


CASE mTxQueueReset OF
	E_CanItfHelperHResult.NoError_11Bit .. E_CanItfHelperHResult.NoError_29Bit_nTrans:
		IF (pTxQueue<>0) THEN
			MEMSET(destAddr := pTxQueue, 0, n :=cbTxQueueSize);
			_nTxMsgSendCnt := 0;
			_bTxMsgSent := FALSE;
			mTxQueueReset := E_CanItfHelperHResult.NoError;
		ELSE
			mTxQueueReset := E_CanItfHelperHResult.InvalidSetup;
		END_IF;
END_CASE
END_METHOD

END_FUNCTION_BLOCK

// Utilities/POUs/F_CanMessage_TO_CSV
{attribute 'hide_all_locals' := ''}
FUNCTION F_CanMessage_TO_CSV : STRING //output -> cobid ,datalength ,extended address ,rtr ,data
VAR_INPUT
	stInput: ST_CanMsg;
END_VAR
VAR
	nPrecision: INT;
	sTemp: STRING;
END_VAR

IF (stInput.CanHeader.bExtendedAddress) THEN
	nPrecision := 8;
ELSE
	nPrecision := 3;
END_IF
 
F_CanMessage_TO_CSV := 	CONCAT('16#',
							CONCAT( DWORD_TO_HEXSTR(stInput.CanHeader.nCobid,nPrecision,FALSE),
								CONCAT(Param_CanItfHelper.sCSV_deliminator,
									CONCAT(UINT_TO_STRING(stInput.CanHeader.nMsgLength),
										CONCAT(Param_CanItfHelper.sCSV_deliminator,
											CONCAT(BOOL_TO_STRING(stInput.CanHeader.bExtendedAddress),
												CONCAT(Param_CanItfHelper.sCSV_deliminator,
													CONCAT(BOOL_TO_STRING(stInput.CanHeader.bRTR),
														CONCAT(Param_CanItfHelper.sCSV_deliminator,
															DATA_TO_HEXSTR(pData := ADR(stInput.CanData), cbData := USINT_TO_UDINT(SIZEOF(stInput.CanData)),bLoCase := FALSE))))))))));

END_FUNCTION

// Utilities/POUs/F_CSV_TO_CanMessage
{attribute 'hide_all_locals'}
FUNCTION F_CSV_TO_CanMessage : ST_CanMsg//input -> cobid ,datalength ,extended address ,rtr ,data
VAR_INPUT
	sInput: STRING;//all four deliminators required
END_VAR
VAR
	//sWorkingValue : STRING;
	nTemp: INT;
	sDelim: STRING;
END_VAR


sInput := F_ToUCase(in:= sInput);

sDelim := Param_CanItfHelper.sCSV_deliminator; 

nTemp := FIND(STR1 := sInput, STR2:= sDelim);
F_CSV_TO_CanMessage.CanHeader.nCobid := STRING_TO_UDINT(LEFT(STR:= sInput,SIZE := nTemp));
sInput :=RIGHT(STR:= sInput, SIZE:= LEN(sInput) - nTemp);

nTemp := FIND(STR1 := sInput, STR2:= sDelim);
F_CSV_TO_CanMessage.CanHeader.nMsgLength :=STRING_TO_UINT(LEFT(STR:= sInput,SIZE := nTemp));
sInput :=RIGHT(STR:= sInput, SIZE:= LEN(sInput) - nTemp);

nTemp := FIND(STR1 := sInput, STR2:= sDelim);
F_CSV_TO_CanMessage.CanHeader.bExtendedAddress :=STRING_TO_BOOL(LEFT(STR:= sInput,SIZE := nTemp));
sInput :=RIGHT(STR:= sInput, SIZE:= LEN(sInput) - nTemp);

nTemp := FIND(STR1 := sInput, STR2:= sDelim);
F_CSV_TO_CanMessage.CanHeader.bRTR :=STRING_TO_BOOL(LEFT(STR:= sInput,SIZE := nTemp));
sInput :=RIGHT(STR:= sInput, SIZE:= LEN(sInput) - nTemp);

HEXSTR_TO_DATA(sHex:=sInput,pData := ADR(F_CSV_TO_CanMessage.CanData), cbData := SIZEOF(F_CSV_TO_CanMessage.CanData));

END_FUNCTION

// Utilities/POUs/FB_RxMapper
{attribute 'hide_all_locals'}
FUNCTION_BLOCK FB_RxMapper //See ST_RxMapping for more info.
VAR_INPUT
	bRun					: BOOL;
	bAutoCreateMappings		: BOOL; //Be careful with this, can quickly cause the Rx Mapper to use a lot of CPU time. This can lead to cycle exceeds. Configure CAN Interface RxFilter is recommeded if used!
	pCanItfHelper 			: POINTER TO FB_CanItfHelper;
	cbCanItfHelperSize		: UDINT; 
	paMappingData 			: POINTER TO ARRAY[0..65535] OF ST_RxMapping;
	cbMappingDataSize		: UDINT;
END_VAR
VAR_OUTPUT
	bBusy 					: BOOL;
	bError					: BOOL;
	eRxMapperHResult 		: E_CanRxMapperHResult;
	nMappingCnt				: UDINT;
END_VAR
VAR
	bUnmappedCanMsg			: BOOL;
	nRxMapperUpperIndex		: UDINT;
	nCobidtemp				: UDINT;
	nPrevRxCounter 			: UINT;
	index 					: UINT;
	stTempCanMsg			: ST_CanMsg;
	nMappingIndex 			: UDINT;
	CanHelperHResult		: E_CanItfHelperHResult;
END_VAR

IF NOT bRun THEN
	bBusy := FALSE;
	RETURN;
ELSE
	bBusy := TRUE;
END_IF

eRxMapperHResult := mCheckSetup();
IF (eRxMapperHResult < 0 ) THEN
	bError := TRUE;
	RETURN;
END_IF

eRxMapperHResult := E_CanRxMapperHResult.NoError;

nRxMapperUpperIndex := (cbMappingDataSize / SIZEOF(ST_RxMapping))-1;

FOR index:=0 TO GVL_CanItfHelper.nRxQueueUpperIndex BY 1 DO
	MEMSET(destAddr := ADR(stTempCanMsg), 0, n:=SIZEOF(stTempCanMsg));
	CanHelperHResult := pCanItfHelper^.mRxMessageGet(bPeakOnly := TRUE, pRxCanMessage := ADR(stTempCanMsg));
	IF CanHelperHResult >= 0 THEN
		bUnmappedCanMsg := TRUE; //used later
		FOR nMappingIndex:= 0 TO MIN(nMappingCnt-1 , nRxMapperUpperIndex) BY 1 DO
			IF (paMappingData^[nMappingIndex].i_stCanMsg.CanHeader.nCobid = stTempCanMsg.CanHeader.nCobid) AND (paMappingData^[nMappingIndex].i_stCanMsg.CanHeader.bExtendedAddress = stTempCanMsg.CanHeader.bExtendedAddress) AND (paMappingData^[nMappingIndex].i_stCanMsg.CanHeader.bRTR = stTempCanMsg.CanHeader.bRTR) THEN
				bUnmappedCanMsg := FALSE;
				IF paMappingData^[nMappingIndex].i_bRun THEN
					IF 	(paMappingData^[nMappingIndex].i_pDestAddr <> 0) AND 
						(paMappingData^[nMappingIndex].i_cbDestSize <> 0) AND 
						(paMappingData^[nMappingIndex].i_cbDestSize >= UINT_TO_UDINT(stTempCanMsg.CanHeader.nMsgLength)) THEN
							paMappingData^[nMappingIndex].i_stCanMsg := stTempCanMsg;
							MEMCPY(paMappingData^[nMappingIndex].i_pDestAddr ,ADR(paMappingData^[nMappingIndex].i_stCanMsg.CanData[0]), paMappingData^[nMappingIndex].i_stCanMsg.CanHeader.nMsgLength);
							paMappingData^[nMappingIndex].o_bBusy := TRUE;
							paMappingData^[nMappingIndex].o_nUpdateCount := paMappingData^[nMappingIndex].o_nUpdateCount +1;					
					ELSE
						paMappingData^[nMappingIndex].o_bError := TRUE;
						eRxMapperHResult := E_CanRxMapperHResult.RxMappingHasError;
					END_IF					
				END_IF
			END_IF
		END_FOR
		IF bUnmappedCanMsg AND bAutoCreateMappings THEN
			eRxMapperHResult := THIS^.mCreateMsgMapping(bRun:=FALSE, stCanMsg:= stTempCanMsg,pDestAddr:= 0, cbDestSize := 0);
		END_IF
	END_IF
END_FOR

METHOD mAddMapping : E_CanRxMapperHResult
VAR_INPUT
	stInput		: ST_RxMapping;
END_VAR
mAddMapping := mCheckSetup();
IF (mAddMapping < 0 ) THEN
	bError := TRUE;
	RETURN;
END_IF

nRxMapperUpperIndex := (cbMappingDataSize / SIZEOF(ST_RxMapping))-1;

IF ((nMappingCnt > nRxMapperUpperIndex) OR (cbMappingDataSize = 0)) THEN
	mAddMapping := E_CanRxMapperHResult.RxMappingsListFull;
	RETURN;
END_IF

IF (stInput.i_bRun = FALSE) THEN
	mAddMapping := E_CanRxMapperHResult.RxMappingNotRunning;
END_IF

IF stInput.i_cbDestSize < stInput.i_stCanMsg.CanHeader.nMsgLength THEN
	mAddMapping := E_CanRxMapperHResult.RxMappingDestSizeError;
END_IF

IF (stInput.i_pDestAddr = 0) THEN
	mAddMapping := E_CanRxMapperHResult.RxMappingDestPointerError;
END_IF

paMappingData^[nMappingCnt] := stInput;
nMappingCnt := nMappingCnt + 1;
END_METHOD

METHOD PRIVATE mCheckSetup : E_CanRxMapperHResult
VAR_INPUT
END_VAR
IF ((cbMappingDataSize = 0) OR (paMappingData = 0)) THEN
	mCheckSetup := E_CanRxMapperHResult.MappingSetupIsInvalid;
	RETURN;
END_IF

IF ((pCanItfHelper = 0) OR (cbCanItfHelperSize <> SIZEOF(FB_CanItfHelper)))  THEN
	bError := TRUE;
	mCheckSetup := E_CanRxMapperHResult.RxMapperHasInvalidSetup;
	RETURN;
END_IF

IF (NOT pCanItfHelper^.bValidSetup) THEN
	mCheckSetup := E_CanRxMapperHResult.RxMapperHasInvalidSetup;
	RETURN;
END_IF
END_METHOD

METHOD mClearMappings : E_CanRxMapperHResult // clears all mappings paMappingData points to. Result always 0 NoError
mClearMappings := mCheckSetup();
IF (mClearMappings < 0 ) THEN
	bError := TRUE;
	RETURN;
END_IF


mClearMappings := E_CanRxMapperHResult.NoError;
MEMSET(destAddr := ADR(paMappingData^), 0 , n:= SIZEOF(cbMappingDataSize)); //Pointer is to an array varaible, which is also a pointer. Clear the array not the array pointer.
nMappingCnt := 0;
END_METHOD

METHOD mCreateMsgMapping : E_CanRxMapperHResult
VAR_INPUT
	bRun: BOOL;
	stCanMsg : ST_CanMsg;
	pDestAddr : POINTER TO BYTE;
	cbDestSize	: UDINT;
END_VAR
VAR
	temp: ST_RxMapping;
END_VAR
mCreateMsgMapping := E_CanRxMapperHResult.NoError;

temp.i_bRun := bRun;
temp.i_stCanMsg := stCanMsg;
temp.i_pDestAddr := pDestAddr;
temp.i_cbDestSize:= cbDestSize;

mCreateMsgMapping := This^.mAddMapping(temp);
END_METHOD

METHOD mCreateNewMapping : E_CanRxMapperHResult
VAR_INPUT
	bRun: BOOL;
	nCobid : DWORD;
	nMsgLength : UINT;
	pDestAddr : POINTER TO BYTE;
	cbDestSize	: UDINT;
END_VAR
VAR
	temp: ST_RxMapping;
END_VAR
mCreateNewMapping := E_CanRxMapperHResult.NoError;

temp.i_bRun := bRun;
temp.i_stCanMsg.CanHeader.nCobid := nCobid;
temp.i_stCanMsg.CanHeader.nMsgLength := nMsgLength;
temp.i_pDestAddr := pDestAddr;
temp.i_cbDestSize:= cbDestSize;

mCreateNewMapping := This^.mAddMapping(temp);
END_METHOD

METHOD mSetMappingCnt : E_CanRxMapperHResult  // return true if successful, must be less then or equal to size of mapping array.
VAR_INPUT
	input : UDINT;
END_VAR
mSetMappingCnt := mCheckSetup();
IF (mSetMappingCnt < 0 ) THEN
	bError := TRUE;
	RETURN;
END_IF

nRxMapperUpperIndex := (cbMappingDataSize / SIZEOF(ST_RxMapping))-1;

IF input > nRxMapperUpperIndex THEN
	nMappingCnt := input;
	mSetMappingCnt := E_CanRxMapperHResult.InvalidParameter;
END_IF
END_METHOD

END_FUNCTION_BLOCK
